Fanuc KAREL source: kb00119.KL

-- PROVISIONAL review KL for V1013-1; original PC SHA256 455c6751c0084e53e5a82ecf70f2ee0416153d7c7301dbb6d53e17dfb4ce124e
-- Incomplete behavior may be omitted. Consult companion uncertainty JSON. Do not deploy.
PROGRAM KB00119
%NOLOCKGROUP
BEGIN
  -- UNRESOLVED_PC offsets 5-12; opcodes 9D,23
  -- UNRESOLVED_PC offsets 17-24; opcodes 9D,23
  -- UNRESOLVED_PC offsets 29-45; opcodes 27,22,22,31
  -- UNRESOLVED_PC offsets 50-54; opcodes 7F
END KB00119
